{attribute 'TcGenerated'}
{attribute 'no-analysis'}
{attribute 'linkalways'}
// This function has been automatically generated from the project information.
VAR_GLOBAL CONSTANT
	{attribute 'const_non_replaced'}
	stLibVersion_TcUnit_verifier : ST_LibVersion := (iMajor := 1, iMinor := 2, iBuild := 1, iRevision := 0, sVersion := '1.2.1.0');
END_VAR

(* stored: Version 1.1.0.1
   GVL Global_Version: Id {9b38d0ad-c87b-4c0f-81f8-641cbe7dcd8c} *)
